	300:
		stAxis[GVL.cXP].mcMoveAbs(Axis:=stAxis[GVL.cXP].axisRef, Execute:=FALSE);
		stAxis[GVL.cXM].mcMoveAbs(Axis:=stAxis[GVL.cXM].axisRef, Execute:=FALSE);
		stAxis[GVL.cXP].mcMoveRel(Axis:=stAxis[GVL.cXP].axisRef, Execute:=FALSE);
		stAxis[GVL.cXM].mcMoveRel(Axis:=stAxis[GVL.cXM].axisRef, Execute:=FALSE);
		stAxis[GVL.cXP].mcJog(Axis:=stAxis[GVL.cXP].axisRef, JogForward:=FALSE, JogBackwards:=FALSE);
		stAxis[GVL.cXM].mcJog(Axis:=stAxis[GVL.cXM].axisRef, JogForward:=FALSE, JogBackwards:=FALSE);
		nNextState := 400;
		
	400:
		stAxis[GVL.cXP].mcReset(axis:=stAxis[GVL.cXP].axisRef, Execute:=TRUE);
		stAxis[GVL.cXM].mcReset(axis:=stAxis[GVL.cXM].axisRef, Execute:=TRUE);
		IF stAxis[GVL.cXP].mcReset.Done AND stAxis[GVL.cXM].mcReset.Done THEN
			stAxis[GVL.cXP].mcReset(axis:=stAxis[GVL.cXP].axisRef, Execute:=FALSE);
			stAxis[GVL.cXM].mcReset(axis:=stAxis[GVL.cXM].axisRef, Execute:=FALSE);
			bResetting := FALSE;
			nNextState := 100;
		END_IF
		//d := d+1;

END_CASE

END_FUNCTION_BLOCK

// ---- POUs/StateMachine/StateTop/FB_StateDisabled.TcPOU
FUNCTION_BLOCK FB_StateDisabled
VAR_IN_OUT
	stAxis  : ARRAY [GVL.cXP .. GVL.cXM] OF ST_AxisGroup;
	bTopentry : BOOL;
END_VAR
VAR_OUTPUT
	nSMState	: DINT;
END_VAR
VAR_INPUT

END_VAR

IF bTopEntry = TRUE THEN
	bTopEntry := FALSE;
END_IF	
	
stAxis[GVL.cXP].mcPower(Axis := stAxis[GVL.cXP].axisRef, Enable_Positive := FALSE, Enable_Negative := FALSE);
stAxis[GVL.cXM].mcPower(Axis := stAxis[GVL.cXM].axisRef, Enable_Positive := FALSE, Enable_Negative := FALSE);	
stAxis[GVL.cXP].mcHome(Axis := stAxis[GVL.cXP].axisRef, Execute := FALSE);
stAxis[GVL.cXM].mcHome(Axis := stAxis[GVL.cXP].axisRef, Execute := FALSE);
stAxis[GVL.cXP].mcReset(Axis := stAxis[GVL.cXP].axisRef, Execute := FALSE);
stAxis[GVL.cXM].mcReset(Axis := stAxis[GVL.cXM].axisRef, Execute := FALSE);
stAxis[GVL.cXP].bBrake 	:= GVL.cBrakeOn;
stAxis[GVL.cXM].bBrake 	:= GVL.cBrakeOn;
GVL.fbWaitTimer(IN:=FALSE);

nSMState := 10000;

END_FUNCTION_BLOCK

// ---- POUs/FB_Power.TcPOU
FUNCTION_BLOCK FB_Power

VAR_IN_OUT
	state : INT;
END_VAR

VAR
	//Power variable
	Vraw AT %I*	: ARRAY [0 .. E_Components.system] OF DINT;
	Vsense		: ARRAY [0 .. E_Components.system] OF REAL;
	Iin			: ARRAY [0 .. E_Components.system] OF REAL;
	Pin		 	: ARRAY [0 .. E_Components.system] OF REAL;
	Pin_max		: ARRAY [0 .. E_Components.system] OF REAL;
	Pin_avg		: ARRAY [0 .. E_Components.system] OF REAL;
	
	//counter
	i 				: INT;
	powerTotal		: ARRAY [0 .. E_Components.system] OF REAL;
	powerCounter 	: ARRAY [0 .. E_Components.system] OF DINT;
	
	//timer
	timer 			: TON;
	timeElapsed		: TIME;
	timer_rtrig		: R_TRIG;
	
	//testvar
	test : INT;
END_VAR

VAR CONSTANT
	Rsense			: REAL := 0.051;
	AdcResolution	: DINT := 8388607; //24bit adc (positive and minus)
	Vin				: ARRAY[0..1] OF REAL := [24.0, 48.0];
	Vref			: REAL := 1.25;
	CountTo			: TIME := T#1000H;
END_VAR

(*This function block is used to monitor shutter system power usage.
The module calculates instantanuous power, average power usage over a motion duration, and max power  *)

//reset power values
IF state=0 THEN
	FOR i := 0 TO E_Components.system BY 1 DO
		Pin_max[i] := 0;
	END_FOR
END_IF


FOR i:=0 TO (E_Components.system - 1) BY 1 DO 

//Calculate instantanuous power
	Vsense[i] := (DINT_TO_REAL(Vraw[i])*Vref)/DINT_TO_REAL(AdcResolution);
	Iin[i] := Vsense[i]/Rsense;
	
	IF i=E_Components.motorXM OR i=E_Components.motorXP THEN
		Pin[i] := Vin[1]*Iin[i];
	ELSE
		Pin[i] := Vin[0]*Iin[i];
	END_IF

	
//Calculate average power
	IF state <> 100 THEN
		powerTotal[i] := powerTotal[i]+Pin[i];
		powerCounter[i] := powerCounter[i]+1;
		Pin_avg[i] 		:= PowerTotal[i]/DINT_TO_REAL(powerCounter[i]);
	ELSE
			powertotal[i] 	:= 0;
			powerCounter[i]	:= 0;	
	END_IF

	
//Calculate max power
	IF Pin_max[i] < Pin[i] THEN
		Pin_max[i] := Pin[i];
	END_IF
	
END_FOR


//Calculate power of entire shutter
Pin[E_Components.system] := Pin[E_Components.motorXP]+Pin[E_Components.motorXM]+Pin[E_Components.brakes]
								+ Pin[E_Components.controller]+Pin[E_Components.terminals];
Pin_avg[E_Components.system] := Pin_avg[E_Components.motorXP]+Pin_avg[E_Components.motorXM]+Pin_avg[E_Components.brakes]
								+ Pin_avg[E_Components.controller]+Pin_avg[E_Components.terminals];
IF Pin_max[E_Components.system] < Pin[E_Components.system] THEN
	Pin_max[E_Components.system] := Pin[E_Components.system];
END_IF

END_FUNCTION_BLOCK

// ---- POUs/FB_Protection.TcPOU
FUNCTION_BLOCK FB_Protection
VAR_IN_OUT
	stAxis  			: ARRAY [GVL.cXP .. GVL.cXM] OF ST_AxisGroup;
	eCommand 			: E_Commands;
	//communication IN
	inCalibrate 		: ST_Calibrate;			// no protection needed
	inChangeAxisEnable	: ST_ChangeAxisEnable;	// no protection needed
	inChangeBrakeState	: ST_ChangeBrakeState;	// no protection needed
	inClearAllFaults	: ST_ClearAllFaults;	// no protection needed
	inClearAxisFaults	: ST_ClearAxisFaults;	// no protection needed
	inCloseShutter		: ST_CloseShutter;		
	inDisableAllAxes	: ST_DisableAllAxes;
	inEnableAllAxes		: ST_EnableAllAxes;
	inGoToProd			: ST_GoToProd;
	inHomeAxis			: ST_HomeAxis;
	inMoveAxisAbsolute	: ST_MoveAxisAbsolute;
	inMoveAxisRelative	: ST_MoveAxisRelative;
	inOpenShutter		: ST_OpenShutter;
	inReset				: ST_Reset;
	inTakeExposure		: ST_TakeExposure;
	inToggleSafetyCheck	: ST_ToggleSafetyCheck;
END_VAR
VAR_INPUT
	nState 			: DINT;
END_VAR
VAR_OUTPUT
	nShutterError	: UINT;
END_VAR
VAR
	checkHomed_TON 	: TON;
	
	//for use end of travel protection
	fEotDistTravel	: ARRAY [GVL.cXP .. GVL.cXM, cLmHome .. cLmDeploy] OF LREAL;
	fEotDistStart	: ARRAY [GVL.cXP .. GVL.cXM, cLmHome .. cLmDeploy] OF LREAL;
	fbEotRtrig		: ARRAY [GVL.cXP .. GVL.cXM, cLmHome .. cLmDeploy] OF R_Trig;
	
	//other Var
	i	: INT;
	bBadHall : BOOL;
END_VAR

VAR CONSTANT
	cLmHome 		: INT 	:= 0;
	cLmDeploy		: INT 	:= 1;
	cEotTravelLm	: LREAL := 1.5;
	cDiffLimit 		: LREAL	:= 5;
	cPosError		: LREAL	:= 0.3;
	cExpoTimer		: TIME	:= T#100MS;
	cMaxVelocity	: LREAL	:= 1668.355556;
	cMinVelocity	: LREAL	:= 0;
END_VAR

(*
This function block contains the logic for the shutter system protection. 
*)
/////////////////////////////////////////////////////////////////////////////////////////////////////////////////////
(*Reset Errors*)
/////////////////////////////////////////////////////////////////////////////////////////////////////////////////////
IF (eCommand=E_Commands.reset) THEN
	stAxis[GVL.cXP].fPosDiffAtTrip 		:= 0;
	stAxis[GVL.cXM].fPosDiffAtTrip 		:= 0;
	fEotDistStart[GVL.cXP,cLmHome] 		:= stAxis[GVL.cXP].axisRef.NcToPlc.ActPos;
	fEotDistStart[GVL.cXP,cLmDeploy] 	:= stAxis[GVL.cXP].axisRef.NcToPlc.ActPos;
	fEotDistStart[GVL.cXM,cLmHome] 		:= stAxis[GVL.cXM].axisRef.NcToPlc.ActPos;
	fEotDistStart[GVL.cXM,cLmDeploy] 	:= stAxis[GVL.cXM].axisRef.NcToPlc.ActPos;
	nShutterError 						:= 0;
END_IF
IF (eCommand=E_Commands.calibrate) THEN
	bBadHall := FALSE;
END_IF

nShutterError.0 := 0;

/////////////////////////////////////////////////////////////////////////////////////////////////////////////////////
(*Check brake status - prevents motion if motion is commanded while brake is engaged*)
/////////////////////////////////////////////////////////////////////////////////////////////////////////////////////
IF stAxis[GVL.cXP].bBrake = GVL.cBrakeOn OR stAxis[GVL.cXM].bBrake = GVL.cBrakeOn THEN
	IF stAxis[GVL.cXP].axisRef.Status.Moving OR stAxis[GVL.cXM].axisRef.Status.Moving THEN
		//////// --set error here-- //////////////////////////////////////////////////////////////////////////////////////////
		nShutterError.1 := 1;
	ELSE
		nShutterError.1 := 0;
	END_IF
END_IF

/////////////////////////////////////////////////////////////////////////////////////////////////////////////////////
(*Check position differences - Compare hall switch and motor encoder position. Stop motion if greater than diffLimit.*)
/////////////////////////////////////////////////////////////////////////////////////////////////////////////////////
IF stAxis[GVL.cXP].bIsCalibrated AND stAxis[GVL.cXM].bIsCalibrated THEN
	IF ABS(stAxis[GVL.cXP].fPosDiffAtTrip)>cDiffLimit OR ABS(stAxis[GVL.cXM].fPosDiffAtTrip)>cDiffLimit THEN
		//////// --set error here-- /////////////////////////////////////////////////////////////////////////////////
		nShutterError.2 := 1;
	ELSE
		nShutterError.2 := 0;
	END_IF
END_IF

/////////////////////////////////////////////////////////////////////////////////////////////////////////////////////
(*Check exposure time - If less than 100 ms, prevent exposure command from running*)
/////////////////////////////////////////////////////////////////////////////////////////////////////////////////////
IF (inTakeExposure.exposureTime<cExpoTimer AND eCommand=E_Commands.takeExposure) THEN
	eCommand := E_Commands.noCommand;
	//////// --set error here-- /////////////////////////////////////////////////////////////////////////////////
	nShutterError.3 := 1;
ELSE
	nShutterError.3 := 0;
END_IF

/////////////////////////////////////////////////////////////////////////////////////////////////////////////////////
(*Check home status - Prevents all other motion if not homed*)
/////////////////////////////////////////////////////////////////////////////////////////////////////////////////////
IF NOT stAxis[GVL.cXP].axisRef.Status.Homed OR NOT stAxis[GVL.cXM].axisRef.Status.Homed THEN
	IF eCommand=E_Commands.closeShutter OR eCommand=E_Commands.goToProd 
		OR eCommand=E_Commands.moveAxisAbsolute OR eCommand=E_Commands.moveAxisRelative 
		OR eCommand=E_Commands.openShutter OR eCommand=E_Commands.takeExposure THEN
			//////// --set error here-- /////////////////////////////////////////////////////////////////////////////////
			nShutterError.4 := 1;
	END_IF
ELSE
	nShutterError.4 := 0;
END_IF
/////////////////////////////////////////////////////////////////////////////////////////////////////////////////////
(*Check for NC errors. If any, disable movement for both motors*)
/////////////////////////////////////////////////////////////////////////////////////////////////////////////////////
IF stAxis[GVL.cXP].axisRef.Status.Error OR stAxis[GVL.cXM].axisRef.Status.Error THEN
	stAxis[GVL.cXP].mcPower(Axis := stAxis[GVL.cXP].axisRef, Enable_Positive := FALSE, Enable_Negative := FALSE);
	stAxis[GVL.cXM].mcPower(Axis := stAxis[GVL.cXM].axisRef, Enable_Positive := FALSE, Enable_Negative := FALSE); 
	stAxis[GVL.cXP].bBrake := GVL.cBrakeOn;
	stAxis[GVL.cXM].bBrake := GVL.cBrakeOn;
	//////// --set error here-- /////////////////////////////////////////////////////////////////////////////////
	nShutterError.5 := 1;
ELSE
	nShutterError.5 := 0;
END_IF

/////////////////////////////////////////////////////////////////////////////////////////////////////////////////////
(*Check calibration status - If one blade set is not calibrated, speed cannot be higher than 200 mms.*)
/////////////////////////////////////////////////////////////////////////////////////////////////////////////////////
IF NOT stAxis[GVL.cXP].bIsCalibrated OR NOT stAxis[GVL.cXM].bIsCalibrated THEN
	IF (inMoveAxisAbsolute.speed>200) THEN
		inMoveAxisAbsolute.speed := 0;
		//////// --set error here-- /////////////////////////////////////////////////////////////////////////////////
		nShutterError.6 := 1;
	END_IF
ELSE
	nShutterError.6:= 0;
END_IF

/////////////////////////////////////////////////////////////////////////////////////////////////////////////////////
(*Check that one blade set cannot be commanded to pass limit*)
/////////////////////////////////////////////////////////////////////////////////////////////////////////////////////
IF (eCommand=E_Commands.moveAxisAbsolute AND (stAxis[GVL.cXP].axisRef.Status.Homed AND stAxis[GVL.cXM].axisRef.Status.Homed)) THEN
	IF (inMoveAxisAbsolute.position<(GVL.cPosStart-cPosError) OR inMoveAxisAbsolute.position>(GVL.cPosEnd+cPosError)) THEN
		eCommand := E_Commands.noCommand;
		//////// --set error here-- /////////////////////////////////////////////////////////////////////////////////
		nShutterError.7 := 1;
	END_IF
END_IF
IF (eCommand=E_Commands.moveAxisRelative AND (stAxis[GVL.cXP].axisRef.Status.Homed AND stAxis[GVL.cXM].axisRef.Status.Homed)) THEN
	IF ((inMoveAxisRelative.distance+stAxis[inMoveAxisRelative.axisIndex].axisRef.NcToPlc.ActPos)<(GVL.cPosStart-cPosError) 
		OR (inMoveAxisRelative.distance+stAxis[inMoveAxisRelative.axisIndex].axisRef.NcToPlc.ActPos)>(GVL.cPosEnd+cPosError)) THEN
		eCommand := E_Commands.noCommand;
		//////// --set error here-- /////////////////////////////////////////////////////////////////////////////////
		nShutterError.7 := 1;
	END_IF
END_IF

/////////////////////////////////////////////////////////////////////////////////////////////////////////////////////
(*Check that one blade set cannot be commanded to pass the other blade set's position*)
/////////////////////////////////////////////////////////////////////////////////////////////////////////////////////
IF (eCommand=E_Commands.moveAxisAbsolute) THEN
	IF (inMoveAxisAbsolute.axisIndex=GVL.cXP AND inMoveAxisAbsolute.position>(stAxis[GVL.cXM].axisRef.NcToPlc.ActPos+cPosError)) THEN
		eCommand := E_Commands.noCommand;
		//////// --set error here-- /////////////////////////////////////////////////////////////////////////////////
		nShutterError.8 := 1;
	END_IF
	IF (inMoveAxisAbsolute.axisIndex=GVL.cXM AND inMoveAxisAbsolute.position<(stAxis[GVL.cXP].axisRef.NcToPlc.ActPos-cPosError)) THEN
		eCommand := E_Commands.noCommand;
		//////// --set error here-- /////////////////////////////////////////////////////////////////////////////////
		nShutterError.8 := 1;
	END_IF
END_IF

IF (eCommand=E_Commands.moveAxisRelative) THEN
	IF (inMoveAxisRelative.axisIndex=GVL.cXP AND (inMoveAxisRelative.distance+stAxis[GVL.cXP].axisRef.NcToPlc.ActPos)>(stAxis[GVL.cXM].axisRef.NcToPlc.ActPos+cPosError)) THEN
		eCommand := E_Commands.noCommand;
		//////// --set error here-- /////////////////////////////////////////////////////////////////////////////////
		nShutterError.8 := 1;
	END_IF
	IF (inMoveAxisRelative.axisIndex=GVL.cXM AND (inMoveAxisRelative.distance+stAxis[GVL.cXM].axisRef.NcToPlc.ActPos)<(stAxis[GVL.cXP].axisRef.NcToPlc.ActPos-cPosError)) THEN
		eCommand := E_Commands.noCommand;
		//////// --set error here-- /////////////////////////////////////////////////////////////////////////////////
		nShutterError.8 := 1;
	END_IF
END_IF

/////////////////////////////////////////////////////////////////////////////////////////////////////////////////////
(* Checks to see if blades have reach end of travel. If it has, stop further motion in that direction	*)
/////////////////////////////////////////////////////////////////////////////////////////////////////////////////////
//End of travel stop
IF(stAxis[GVL.cXP].axisRef.Status.Homed AND stAxis[GVL.cXM].axisRef.Status.Homed) THEN
	fbEotRtrig[GVL.cXP,cLmHome](CLK := stAxis[GVL.cXP].bLimitHome);
	fbEotRtrig[GVL.cXP,cLmDeploy](CLK := stAxis[GVL.cXP].bLimitDeployed);
	fbEotRtrig[GVL.cXM,cLmHome](CLK := stAxis[GVL.cXM].bLimitHome);
	fbEotRtrig[GVL.cXM,cLmDeploy](CLK := stAxis[GVL.cXM].bLimitDeployed);
	IF fbEotRtrig[GVL.cXP,cLmHome].Q THEN
		fEotDistStart[GVL.cXP,cLmHome] := stAxis[GVL.cXP].axisRef.NcToPlc.ActPos;
	END_IF
	IF fbEotRtrig[GVL.cXP,cLmDeploy].Q THEN
		fEotDistStart[GVL.cXP,cLmDeploy] := stAxis[GVL.cXP].axisRef.NcToPlc.ActPos;
	END_IF
	IF fbEotRtrig[GVL.cXM,cLmHome].Q THEN
		fEotDistStart[GVL.cXM,cLmHome] := stAxis[GVL.cXM].axisRef.NcToPlc.ActPos;
	END_IF
	IF fbEotRtrig[GVL.cXM,cLmDeploy].Q THEN
		fEotDistStart[GVL.cXM,cLmDeploy] := stAxis[GVL.cXM].axisRef.NcToPlc.ActPos;
	END_IF									
	
	IF stAxis[GVL.cXP].bLimitHome THEN
		fEotDistTravel[GVL.cXP,cLmHome] := fEotDistStart[GVL.cXP,cLmHome] - stAxis[GVL.cXP].axisRef.NcToPlc.ActPos;
		IF fEotDistTravel[GVL.cXP,cLmHome] > cEotTravelLm THEN
			stAxis[GVL.cXP].mcPower(Axis := stAxis[GVL.cXP].axisRef, Enable_Negative := FALSE);
		END_IF
	END_IF
	
	IF stAxis[GVL.cXP].bLimitDeployed THEN
		fEotDistTravel[GVL.cXP,cLmDeploy] := stAxis[GVL.cXP].axisRef.NcToPlc.ActPos - fEotDistStart[GVL.cXP,cLmDeploy];
		IF fEotDistTravel[GVL.cXP,cLmHome] > cEotTravelLm THEN
			stAxis[GVL.cXP].mcPower(Axis := stAxis[GVL.cXP].axisRef, Enable_Positive := FALSE);
		END_IF
	END_IF
	
	IF stAxis[GVL.cXM].bLimitHome THEN
		fEotDistTravel[GVL.cXM,clmHome] := stAxis[GVL.cXM].axisRef.NcToPlc.ActPos - fEotDistStart[GVL.cXM,cLmHome];
		IF fEotDistTravel[GVL.cXM,cLmHome] > cEotTravelLm THEN
			stAxis[GVL.cXM].mcPower(Axis := stAxis[GVL.cXM].axisRef, Enable_Positive := FALSE);
		END_IF
	END_IF
	
	IF stAxis[GVL.cXM].bLimitDeployed THEN
		fEotDistTravel[GVL.cXM,cLmDeploy] := fEotDistStart[GVL.cXM,cLmDeploy] - stAxis[GVL.cXM].axisRef.NcToPlc.ActPos;
		IF fEotDistTravel[GVL.cXM,cLmHome] > cEotTravelLm THEN
			stAxis[GVL.cXM].mcPower(Axis := stAxis[GVL.cXM].axisRef, Enable_Negative := FALSE);
		END_IF
	END_IF
END_IF

/////////////////////////////////////////////////////////////////////////////////////////////////////////////////////
(* if hall signal changes during no motion, system needs to recalibrate	*)
/////////////////////////////////////////////////////////////////////////////////////////////////////////////////////
FOR i:=GVL.cHallLower TO GVL.cHallUpper BY 1 DO
	IF GVL.nNumOfInputs[i].0 AND ((NOT stAxis[GVL.cXP].axisRef.Status.Moving) AND (NOT stAxis[GVL.cXM].axisRef.Status.Moving)) THEN
		bBadHall := TRUE;
	END_IF
END_FOR
IF bBadHall THEN
	IF eCommand=E_Commands.closeShutter OR eCommand=E_Commands.goToProd 
		OR eCommand=E_Commands.moveAxisAbsolute OR eCommand=E_Commands.moveAxisRelative 
		OR eCommand=E_Commands.openShutter OR eCommand=E_Commands.takeExposure THEN
			nShutterError.13 := 1;
	END_IF
END_IF

/////////////////////////////////////////////////////////////////////////////////////////////////////////////////////
(* shutter system error handle	*)
/////////////////////////////////////////////////////////////////////////////////////////////////////////////////////

IF (nShutterError.0 OR_ELSE nShutterError.1 OR_ELSE nShutterError.2 OR_ELSE nShutterError.3 OR_ELSE nShutterError.4 OR_ELSE nShutterError.5) THEN
	stAxis[GVL.cXP].mcStop(Axis := stAxis[GVL.cXP].axisRef, Deceleration := 29630, Jerk := 263374.5, Execute := TRUE);
	stAxis[GVL.cXM].mcStop(Axis := stAxis[GVL.cXM].axisRef, Deceleration := 29630, Jerk := 263374.5, Execute := TRUE);
	//stAxis[GVL.cXP].mcPower(Axis := stAxis[GVL.cXP].axisRef, Enable_Positive := FALSE, Enable_Negative := FALSE);
	//stAxis[GVL.cXM].mcPower(Axis := stAxis[GVL.cXM].axisRef, Enable_Positive := FALSE, Enable_Negative := FALSE); 
	IF (nShutterError.0 OR_ELSE nShutterError.2 OR_ELSE nShutterError.3 OR_ELSE nShutterError.4 OR_ELSE nShutterError.5 OR_ELSE nShutterError.13) THEN
		stAxis[GVL.cXP].bBrake := GVL.cBrakeOn;
		stAxis[GVL.cXM].bBrake := GVL.cBrakeOn;
	END_IF
ELSE
	stAxis[GVL.cXP].mcStop(Axis := stAxis[GVL.cXP].axisRef, Execute := FALSE);
	stAxis[GVL.cXM].mcStop(Axis := stAxis[GVL.cXM].axisRef, Execute := FALSE);
END_IF

/////////////////////////////////////////////////////////////////////////////////////////////////////////////////////
(* Other shutter protection	*)
/////////////////////////////////////////////////////////////////////////////////////////////////////////////////////

//Min and Max speed for PROD
IF (inReset.speed>cMaxVelocity) THEN
	inReset.speed:=cMaxVelocity;
ELSIF (inReset.speed<cMinVelocity) THEN
	inReset.speed:=cMinVelocity;
END_IF
//Min and Max speed for move absolute
IF (inMoveAxisAbsolute.speed>cMaxVelocity) THEN
	inReset.speed:=cMaxVelocity;
ELSIF (inMoveAxisAbsolute.speed<cMinVelocity) THEN
	inReset.speed:=cMinVelocity;
END_IF

END_FUNCTION_BLOCK

// ---- POUs/StateMachine/FB_Tracking.TcPOU
FUNCTION_BLOCK FB_Tracking
VAR_IN_OUT
	stAxis  : ARRAY [GVL.cXP .. GVL.cXM] OF ST_AxisGroup;	
END_VAR
VAR_INPUT
	eCommand 			: E_Commands;
	bMotionDone			: BOOL;
	inReset				: ST_Reset;
	inMoveAxisAbsolute	: ST_MoveAxisAbsolute;
	inMoveAxisRelative	: ST_MoveAxisRelative;
END_VAR
VAR_OUTPUT
	stOutMotionDone : ST_MotionDone;
END_VAR
VAR
	//used in tracking Action
	stTrack			: ARRAY [0 .. 4] OF ST_TRACK;
	stTrackTemp		: ST_TRACK;  // Used for the sorting of stTrack.
	keepSorting		: BOOL;      // Used for the sorting.
	bGoNextSeq		: BOOL;
	nAxisID			: INT;
	nMask			: ULINT := 16#FFFF_FFFF_0000_0000;
	
	//used in determining target duration
	fSpeed			: LREAL;
	tTargetDur		: LTIME;
	fDistance		: LREAL;
	
	fbMoving_Rtrig : ARRAY[0 .. 1] OF R_TRIG;
	fbRtrig		: ARRAY[GVL.cHallLower..GVL.cHallUpper] OF R_Trig;
	bInMotion	: BOOL;
	stMotionDone : ARRAY [0..1] OF ST_MotionDone;	
	nSequence	: DINT;
	nLastMoved	: INT;
	
	//counter
	i, j, k, m		: INT := 0;
	nTPC	: INT; //Trip Per Cycle

	// Save task-start and MIO SysTime values in a ring buffer x of depth N. The newest
	// entry is x[i], the oldest is x[(i + 1) mod N], assuming that the buffer is full.
	iTimeBuffer: INT := GVL.cTimeBufferDepth - 1;
	taskStartExtTime: T_TaskStartTimes;
	mioSysTime: T_MioSysTimes;

END_VAR

//////////////////////////////////////////////////////////////
// Call this function block once per cycle to process any updated information about blade set motion and send updates to CCS if required.
//////////////////////////////////////////////////////////////

// Update some times for the previous and current cycles.
iTimeBuffer := (iTimeBuffer + 1) MOD GVL.cTimeBufferDepth;
taskStartExtTime[iTimeBuffer] := F_GetCurExtTime64(GVL.DcToExtTimeOffset, GVL.DcToTcTimeOffset);
mioSysTime[iTimeBuffer] := GVL.mioSysTime;

stAxis[GVL.cXP].bTrackedFlag:=FALSE;
stAxis[GVL.cXM].bTrackedFlag:=FALSE;
nTPC:=0;

// Detect start of motion for the +X blade set, rising edge of its Moving flag from the motor controller.
// Reset motion profile parameters in a local motion-done message not monitored by CCS.
fbMoving_Rtrig[GVL.cXP](CLK:=stAxis[GVL.cXP].axisRef.Status.Moving);
IF fbMoving_Rtrig[GVL.cXP].Q THEN
	// Prepare to record motion profile information.
	bInMotion:=TRUE;  // We're moving!
	stMotionDone[GVL.cXP].axisNum := GVL.cXP; // Axis is +X.
	stMotionDone[GVL.cXP].nsamples := 0;      // No encoder samples yet.
	stMotionDone[GVL.cXP].ntrans := 0;        // No Hall transitions yet.
	stMotionDone[gvl.cXP].startPos := stAxis[GVL.cXP].axisRef.NcToPlc.ActPos;   // Where are we now?
	stMotionDone[GVL.cXP].startTime := taskStartExtTime[iTimeBuffer];
	stMotionDone[GVL.cXP].targetDur := LTIME#0D0H0M0S0MS0US0NS;  // Don't know yet how long this motion will take.
END_IF

// The same, but for the -X blade set.
fbMoving_Rtrig[GVL.cXM](CLK:=stAxis[GVL.cXM].axisRef.Status.Moving);
IF fbMoving_Rtrig[GVL.cXM].Q THEN
	// Prepare to record motion profile information.
	bInMotion:=TRUE;
	stMotionDone[gvl.cXM].axisNum := GVL.cXM;
	stMotionDone[gvl.cXM].nsamples := 0;
	stMotionDone[gvl.cXM].ntrans := 0;
	stMotionDone[gvl.cXM].startPos := stAxis[GVL.cXM].axisRef.NcToPlc.ActPos;
	stMotionDone[gvl.cXM].startTime := taskStartExtTime[iTimeBuffer];
	stMotionDone[gvl.cXM].targetDur := LTIME#0D0H0M0S0MS0US0NS;
END_IF

// Assuming that a motion command was issued by CCS, calculate how long the motion is supposed to last.
// Output is tTargetDur.
IF eCommand = E_Commands.takeExposure THEN
	fSpeed	:= inReset.speed;   // Speed from reset command (actually now set elsewhere in this PLC code).
	IF (fSpeed>0) THEN
		IF (fSpeed>1668.355556) THEN
			fSpeed:=1668.355556;
		END_IF
		tTargetDur 	:= LREAL_TO_LTIME((2*GVL.cPosEnd)/(fSpeed)*EXPT(10,9));
	END_IF
ELSIF eCommand = E_Commands.moveAxisAbsolute THEN
	// MoveAxisAbsolute message contains target position and speed of motion.
	fDistance := ABS(stAxis[inMoveAxisAbsolute.axisIndex].axisRef.NcToPlc.ActPos - inMoveAxisAbsolute.position);
	fSpeed	:= inMoveAxisAbsolute.speed;
	IF (fSpeed>0) THEN
		IF (fSpeed>1668.355556) THEN
			fSpeed:=1668.355556;
		END_IF
		tTargetDur 	:= LREAL_TO_LTIME(((2*fDistance)/(fSpeed))*EXPT(10,9));
	END_IF
ELSIF eCommand = E_Commands.moveAxisRelative THEN
	// MoveAxisRelative message contains position change and how long to take to do it.
	tTargetDur	:= TIME_TO_LTIME(inMoveAxisRelative.moveTime);
END_IF

//Checks to see which blade set last started moving.
IF (stAxis[GVL.cXM].axisRef.Status.Moving AND stAxis[GVL.cXP].axisRef.Status.InTargetPosition) THEN
	nLastMoved:=GVL.cXM;
ELSIF (stAxis[GVL.cXP].axisRef.Status.Moving AND stAxis[GVL.cXM].axisRef.Status.InTargetPosition) THEN
	nLastMoved:=GVL.cXP;
END_IF

////////// Handle the completion of a blade set motion. //////////
IF bMotionDone THEN
	//use for determining which blade set has finished during a travelling slit motion
	IF (stAxis[GVL.cXM].axisRef.Status.Moving AND stAxis[GVL.cXP].axisRef.Status.InTargetPosition) THEN
		nAxisID:=GVL.cXP;
	ELSIF (stAxis[GVL.cXP].axisRef.Status.Moving AND stAxis[GVL.cXM].axisRef.Status.InTargetPosition) THEN
		nAxisID:=GVL.cXM;
	ELSE 
		nAxisID:=nLastMoved;
	END_IF
	//bInMotion flag remains true if either of the blade sets is still in motion
	IF ((NOT stAxis[GVL.cXP].axisRef.Status.Moving) AND (NOT stAxis[GVL.cXM].axisRef.Status.Moving)) THEN
		bInMotion := FALSE;
	END_IF
	// Complete our local motion-done message.
	nSequence := nSequence+1;
	// The motor controller doesn't report exactly when motion was completed, so we assume that it was when the process data
	// from the controller reached us, i.e., at the start of the current cycle.
	stMotionDone[nAxisID].actualDur := ULINT_TO_LTIME(taskStartExtTime[iTimeBuffer] - stMotionDone[nAxisID].startTime);
	stMotionDone[nAxisID].targetDur := tTargetDur;
	stMotionDone[nAxisID].targetPos := stAxis[nAxisID].axisRef.NcToPlc.TargetPos;
	stMotionDone[nAxisID].endPos := stAxis[nAxisID].axisRef.NcToPlc.ActPos;
	stMotionDone[nAxisId].ptpState := MAIN.ptpDiagInfo.PTPState;
	stMotionDone[nAxisId].leapSeconds := MAIN.ptpDiagInfo.CurrentUtcOffset;
	stMotionDone[nAxisId].leapIsValid := TO_BOOL(MAIN.ptpDiagInfo.CurrentUtcOffsetIsValid);
	// Copy our local motion-done message to the location that's monitored by CCS.
	stOutMotionDone:=stMotionDone[nAxisID];
	stOutMotionDone.sequence:=nSequence;  // Ensure message gets sent to CCS by making sure that at least one field has a changed value.
END_IF


////////// Collect information on any Hall switch transitions from the MIOs. //////////
// nNumOfINputs[i] is linked to the event count for the MIO channel assigned to Hall sensor i.
// bInputEventState[i] is linked to the current MIO channel state for Hall sensor i.
// nInputEventTime[i] is linked to the first transition timestamp for Hall sensor i. We assume there is at most one per cycle per channel, though
// more than one channel may have a timestamp available in the same cycle.
// New timestamps are added to the end of the stTrack array.

FOR i:=GVL.cHallLower TO GVL.cHallUpper BY 1 DO
	fbRtrig[i](CLK:=GVL.nNumOfInputs[i].0);  // Look for a rising edge in channel status, which means we have a transition timestamp.
	IF fbRtrig[i].Q THEN
		stTrack[nTPC].nSeqToCompare := INT_TO_WORD((i*10)+5);
		stTrack[nTPC].bEdgeToCompare := GVL.bInputEventState[i];
		stTrack[nTPC].nHallID := i;
		stTrack[nTPC].tScanTime := 
			F_MioExtTime(i, GVL.nInputEventTime[i], iTimeBuffer, taskStartExtTime, mioSysTime);  // ADC timestamp -> ext time.
 		// Count the number of entries stored in stTrack.
		nTPC:=nTPC+1;
	END_IF
END_FOR
	
// Calibration stores events in time order, and later code that assigns locations to Hall events requires
// exactly the same ordering for a given blade set and direction of motion. If during this cycle we picked up
// events from more than one channel we'll have to sort them by time. At most a handful of events
// may occur in a cycle so an exchange sort will do.
IF nTPC > 1 THEN
	keepSorting := TRUE;  // Do we need to keep sorting?
	WHILE keepSorting DO
		keepSorting := FALSE;
		FOR j:= nTPC - 1 TO 1 BY -1 DO
			IF (stTrack[j].tScanTime < stTrack[j-1].tScanTime) THEN  // Use <, not <=, to make it a stable sort.
				stTrackTemp := stTrack[j];
				stTrack[j] := stTrack[j-1];
				stTrack[j-1] := stTrackTemp;
				keepSorting := TRUE;  // Need to keep sorting if an exchange was made.
			END_IF
		END_FOR
	END_WHILE
END_IF


// If we picked up some Hall transitions this cycle, then we need to take position samples (encoder readout).
// We want to check if the position of a blade set at the time of a Hall transition agrees with the
// Hall switch position taken from the last calibration.
IF nTPC>0 THEN
	FOR k:=0 TO nTPC-1 BY 1 DO
		IF (stAxis[GVL.cXP].axisRef.Status.Moving AND stAxis[GVL.cXM].axisRef.Status.Moving) AND
			(stAxis[GVL.cXP].axisRef.Status.PositiveDirection AND stAxis[GVL.cXM].axisRef.Status.PositiveDirection) THEN
			ACT_TrackingDoublePositive();
		ELSIF (stAxis[GVL.cXP].axisRef.Status.Moving AND stAxis[GVL.cXM].axisRef.Status.Moving) AND
			(stAxis[GVL.cXP].axisRef.Status.NegativeDirection AND stAxis[GVL.cXM].axisRef.Status.NegativeDirection) THEN
			ACT_TrackingDoubleNegative();
		ELSE
			ACT_TrackingSingle();
		END_IF
		bGoNextSeq:=FALSE;
	END_FOR
END_IF

ACTION ACT_TrackingDoubleNegative:
// Take encoder samples and compare against Hall transitions when both blade sets are moving toward decreasing camera X coordinate.
// Remember, this code is being called from inside a loop over the contents of stTrack[] with k being the loop variable.
// We have to first assign a Hall event to a blade set before we can find out the motion start times and
// calculate elapsed times from that. 

// +X blade set
IF stAxis[GVL.cXP].axisRef.Status.Moving THEN
	//Compare current sequence with recorded sequence. Update position if match. Negative direction.
	IF stAxis[GVL.cXP].axisRef.status.NegativeDirection AND stAxis[GVL.cXP].stHall[GVL.cDirNeg, stAxis[GVL.cXP].nTripCount].nSeq = stTrack[k].nSeqToCompare AND
			stAxis[GVL.cXP].stHall[GVL.cDirNeg, stAxis[GVL.cXP].nTripCount].bEdge = stTrack[k].bEdgeToCompare AND (NOT bGoNextSeq) THEN
		stAxis[GVL.cXP].fHallPosAct := stAxis[GVL.cXP].fHallPosCal[GVL.cDirNeg, stAxis[GVL.cXP].nTripCount];
		stAxis[GVL.cXP].nTripCount := stAxis[GVL.cXP].nTripCount - 1;		
		//track difference between hall sensor and encoder data at trip point
		stAxis[GVL.cXP].fPosDiffAtTrip := stAxis[GVL.cXP].axisRef.NcToPlc.ActPos - stAxis[GVL.cXP].fHallPosAct;
		stAxis[GVL.cXP].bTrackedFlag:=TRUE;
		bGoNextSeq:=TRUE;
		
		IF bInMotion AND MAIN.outShutterStatus.smState<>E_StatesMaint.Calibrating THEN
			nAxisID := GVL.cXP;
			// The Hall event belongs to the +X blade set.
			stMotionDone[GVL.cXP].trans[stMotionDone[GVL.cXP].ntrans].extTime := stTrack[k].tScanTime;
			stMotionDone[GVL.cXP].trans[stMotionDone[GVL.cXP].ntrans].id := stTrack[k].nHallID;
			stMotionDone[GVL.cXP].trans[stMotionDone[GVL.cXP].ntrans].on := stTrack[k].bEdgeToCompare;
			stMotionDone[GVL.cXP].trans[stMotionDone[GVL.cXP].ntrans].pos := stAxis[GVL.cXP].fHallPosAct;
			stMotionDone[GVL.cXP].ntrans := stMotionDone[GVL.cXP].ntrans +1;
			// We're taking the encoder value from process data for this cycle, so the closest
			// approximation we have to the actual sample time is the time at the start of the cycle.
			stMotionDone[GVL.cXP].samples[stMotionDone[GVL.cXP].nsamples].extTime := taskStartExtTime[iTimeBuffer];
			stMotionDone[GVL.cXP].samples[stMotionDone[GVL.cXP].nsamples].pos := stAxis[GVL.cXP].axisRef.NcToPlc.ActPos;
			stMotionDone[GVL.cXP].nsamples := stMotionDone[GVL.cXP].nsamples + 1;
		END_IF
		
	END_IF
END_IF

// -X blade set
IF stAxis[GVL.cXM].axisRef.Status.Moving THEN
	//Compare current sequence with recorded sequence. Update position if match. Negative direction.
	IF stAxis[GVL.cXM].axisRef.status.NegativeDirection AND stAxis[GVL.cXM].stHall[GVL.cDirNeg, stAxis[GVL.cXM].nTripCount].nSeq = stTrack[k].nSeqToCompare AND
			stAxis[GVL.cXM].stHall[GVL.cDirNeg, stAxis[GVL.cXM].nTripCount].bEdge = stTrack[k].bEdgeToCompare AND (NOT bGoNextSeq) THEN
		stAxis[GVL.cXM].fHallPosAct := stAxis[GVL.cXM].fHallPosCal[GVL.cDirNeg, stAxis[GVL.cXM].nTripCount];
		stAxis[GVL.cXM].nTripCount := stAxis[GVL.cXM].nTripCount + 1;	
		//track difference between hall sensor and encoder data at trip point
		stAxis[GVL.cXM].fPosDiffAtTrip := stAxis[GVL.cXM].axisRef.NcToPlc.ActPos - stAxis[GVL.cXM].fHallPosAct;
		stAxis[GVL.cXM].bTrackedFlag:=TRUE;
		bGoNextSeq:=TRUE;
		
		IF bInMotion AND MAIN.outShutterStatus.smState<>E_StatesMaint.Calibrating THEN
			nAxisID:= GVL.cXM;
			// The Hall event belongs to the -X blade set.
			stMotionDone[GVL.cXM].trans[stMotionDone[GVL.cXM].ntrans].extTime := stTrack[k].tScanTime;
			stMotionDone[GVL.cXM].trans[stMotionDone[GVL.cXM].ntrans].id := stTrack[k].nHallID;
			stMotionDone[GVL.cXM].trans[stMotionDone[GVL.cXM].ntrans].on := stTrack[k].bEdgeToCompare;
			stMotionDone[GVL.cXM].trans[stMotionDone[GVL.cXM].ntrans].pos := stAxis[GVL.cXM].fHallPosAct;
			stMotionDone[GVL.cXM].ntrans := stMotionDone[GVL.cXM].ntrans +1;

			stMotionDone[GVL.cXM].samples[stMotionDone[GVL.cXM].nsamples].extTime := taskStartExtTime[iTimeBuffer];
			stMotionDone[GVL.cXM].samples[stMotionDone[GVL.cXM].nsamples].pos := stAxis[GVL.cXM].axisRef.NcToPlc.ActPos;
			stMotionDone[GVL.cXM].nsamples := stMotionDone[GVL.cXM].nsamples + 1;
		END_IF
		
	END_IF
END_IF
END_ACTION

ACTION ACT_TrackingDoublePositive:
// Take encoder samples and compare against Hall transitions when both blade sets are moving toward increasing camera X coordinate.

// -X blade set
IF stAxis[GVL.cXM].axisRef.Status.Moving THEN
	//Compare current sequence with recorded sequence. Update position if match. Positive direction.
	IF stAxis[GVL.cXM].axisRef.status.PositiveDirection AND stAxis[GVL.cXM].stHall[GVL.cDirPos, stAxis[GVL.cXM].nTripCount].nSeq = stTrack[k].nSeqToCompare AND
			stAxis[GVL.cXM].stHall[GVL.cDirPos, stAxis[GVL.cXM].nTripCount].bEdge = stTrack[k].bEdgeToCompare AND (NOT bGoNextSeq) THEN
		stAxis[GVL.cXM].fHallPosAct := stAxis[GVL.cXM].fHallPosCal[GVL.cDirPos, stAxis[GVL.cXM].nTripCount];
		stAxis[GVL.cXM].nTripCount := stAxis[GVL.cXM].nTripCount - 1;	
		//track difference between hall sensor and encoder data at trip point
		stAxis[GVL.cXM].fPosDiffAtTrip := stAxis[GVL.cXM].axisRef.NcToPlc.ActPos - stAxis[GVL.cXM].fHallPosAct;
		stAxis[GVL.cXM].bTrackedFlag:=TRUE;
		bGoNextSeq:=TRUE;
		
		IF bInMotion AND MAIN.outShutterStatus.smState<>E_StatesMaint.Calibrating THEN
			nAxisID:= GVL.cXM;
			// The Hall event belongs to the -X blade set.
			stMotionDone[GVL.cXM].trans[stMotionDone[GVL.cXM].ntrans].extTime := stTrack[k].tScanTime;
			stMotionDone[GVL.cXM].trans[stMotionDone[GVL.cXM].ntrans].id := stTrack[k].nHallID;
			stMotionDone[GVL.cXM].trans[stMotionDone[GVL.cXM].ntrans].on := stTrack[k].bEdgeToCompare;
			stMotionDone[GVL.cXM].trans[stMotionDone[GVL.cXM].ntrans].pos := stAxis[GVL.cXM].fHallPosAct;
			stMotionDone[GVL.cXM].ntrans := stMotionDone[GVL.cXM].ntrans +1;
			
			stMotionDone[GVL.cXM].samples[stMotionDone[GVL.cXM].nsamples].extTime := taskStartExtTime[iTimeBuffer];
			stMotionDone[GVL.cXM].samples[stMotionDone[GVL.cXM].nsamples].pos := stAxis[GVL.cXM].axisRef.NcToPlc.ActPos;
			stMotionDone[GVL.cXM].nsamples := stMotionDone[GVL.cXM].nsamples + 1;
		END_IF
		
	END_IF
END_IF

// +X blade set
IF stAxis[GVL.cXP].axisRef.Status.Moving THEN
	//Compare current sequence with recorded sequence. Update position if match. Positive direction.
	IF stAxis[GVL.cXP].axisRef.status.PositiveDirection AND stAxis[GVL.cXP].stHall[GVL.cDirPos, stAxis[GVL.cXP].nTripCount].nSeq = stTrack[k].nSeqToCompare AND 
			stAxis[GVL.cXP].stHall[GVL.cDirPos, stAxis[GVL.cXP].nTripCount].bEdge = stTrack[k].bEdgeToCompare AND (NOT bGoNextSeq) THEN
		stAxis[GVL.cXP].fHallPosAct := stAxis[GVL.cXP].fHallPosCal[GVL.cDirPos, stAxis[GVL.cXP].nTripCount];
		stAxis[GVL.cXP].nTripCount := stAxis[GVL.cXP].nTripCount + 1;
		//track difference between hall sensor and encoder data at trip point
		stAxis[GVL.cXP].fPosDiffAtTrip := stAxis[GVL.cXP].axisRef.NcToPlc.ActPos - stAxis[GVL.cXP].fHallPosAct;
		stAxis[GVL.cXP].bTrackedFlag:=TRUE;
		bGoNextSeq:=TRUE;
		
		IF bInMotion AND MAIN.outShutterStatus.smState<>E_StatesMaint.Calibrating THEN
			nAxisID:= GVL.cXP;
			// The Hall event belongs to the +X blade set.
			stMotionDone[GVL.cXP].trans[stMotionDone[GVL.cXP].ntrans].extTime := stTrack[k].tScanTime;
			stMotionDone[GVL.cXP].trans[stMotionDone[GVL.cXP].ntrans].id := stTrack[k].nHallID;
			stMotionDone[GVL.cXP].trans[stMotionDone[GVL.cXP].ntrans].on := stTrack[k].bEdgeToCompare;
			stMotionDone[GVL.cXP].trans[stMotionDone[GVL.cXP].ntrans].pos := stAxis[GVL.cXP].fHallPosAct;
			stMotionDone[GVL.cXP].ntrans := stMotionDone[GVL.cXP].ntrans +1;
			
			// We're taking the encoder value from process data for this cycle, so the closest
			// approximation we have to the actual sample time is the time at the start of the cycle.
			stMotionDone[GVL.cXP].samples[stMotionDone[GVL.cXP].nsamples].extTime := taskStartExtTime[iTimeBuffer];
			stMotionDone[GVL.cXP].samples[stMotionDone[GVL.cXP].nsamples].pos := stAxis[GVL.cXP].axisRef.NcToPlc.ActPos;
			stMotionDone[GVL.cXP].nsamples := stMotionDone[GVL.cXP].nsamples + 1;
		END_IF
		
	END_IF
END_IF
END_ACTION

ACTION ACT_TrackingSingle:
// Take encoder samples and compare against Hall transitions when only one blade set is moving.

// +X blade set
IF stAxis[GVL.cXP].axisRef.Status.Moving THEN
	//Compare current sequence with recorded sequence. Update position if match. Positive direction.
	IF stAxis[GVL.cXP].axisRef.status.PositiveDirection AND stAxis[GVL.cXP].stHall[GVL.cDirPos, stAxis[GVL.cXP].nTripCount].nSeq = stTrack[k].nSeqToCompare AND 
			stAxis[GVL.cXP].stHall[GVL.cDirPos, stAxis[GVL.cXP].nTripCount].bEdge = stTrack[k].bEdgeToCompare AND (NOT bGoNextSeq) THEN
		stAxis[GVL.cXP].fHallPosAct := stAxis[GVL.cXP].fHallPosCal[GVL.cDirPos, stAxis[GVL.cXP].nTripCount];
		stAxis[GVL.cXP].nTripCount := stAxis[GVL.cXP].nTripCount + 1;
		//track difference between hall sensor and encoder data at trip point
		stAxis[GVL.cXP].fPosDiffAtTrip := stAxis[GVL.cXP].axisRef.NcToPlc.ActPos - stAxis[GVL.cXP].fHallPosAct;
		stAxis[GVL.cXP].bTrackedFlag:=TRUE;
		bGoNextSeq:=TRUE;
		
		IF bInMotion AND MAIN.outShutterStatus.smState<>E_StatesMaint.Calibrating THEN
			nAxisID:= GVL.cXP;
			// The Hall event belongs to the +X blade set.
			stMotionDone[GVL.cXP].trans[stMotionDone[GVL.cXP].ntrans].extTime := stTrack[k].tScanTime;
			stMotionDone[GVL.cXP].trans[stMotionDone[GVL.cXP].ntrans].id := stTrack[k].nHallID;
			stMotionDone[GVL.cXP].trans[stMotionDone[GVL.cXP].ntrans].on := stTrack[k].bEdgeToCompare;
			stMotionDone[GVL.cXP].trans[stMotionDone[GVL.cXP].ntrans].pos := stAxis[GVL.cXP].fHallPosAct;
			stMotionDone[GVL.cXP].ntrans := stMotionDone[GVL.cXP].ntrans +1;			
			// We're taking the encoder value from process data for this cycle, so the closest
			// approximation we have to the actual sample time is the time at the start of the cycle.
			stMotionDone[GVL.cXP].samples[stMotionDone[GVL.cXP].nsamples].extTime := taskStartExtTime[iTimeBuffer];
			stMotionDone[GVL.cXP].samples[stMotionDone[GVL.cXP].nsamples].pos := stAxis[GVL.cXP].axisRef.NcToPlc.ActPos;
			stMotionDone[GVL.cXP].nsamples := stMotionDone[GVL.cXP].nsamples + 1;
		END_IF
		
	END_IF
	//Compare current sequence with recorded sequence. Update position if match. Negative direction.
	IF stAxis[GVL.cXP].axisRef.status.NegativeDirection AND stAxis[GVL.cXP].stHall[GVL.cDirNeg, stAxis[GVL.cXP].nTripCount].nSeq = stTrack[k].nSeqToCompare AND
			stAxis[GVL.cXP].stHall[GVL.cDirNeg, stAxis[GVL.cXP].nTripCount].bEdge = stTrack[k].bEdgeToCompare AND (NOT bGoNextSeq) THEN
		stAxis[GVL.cXP].fHallPosAct := stAxis[GVL.cXP].fHallPosCal[GVL.cDirNeg, stAxis[GVL.cXP].nTripCount];
		stAxis[GVL.cXP].nTripCount := stAxis[GVL.cXP].nTripCount - 1;		
		//track difference between hall sensor and encoder data at trip point
		stAxis[GVL.cXP].fPosDiffAtTrip := stAxis[GVL.cXP].axisRef.NcToPlc.ActPos - stAxis[GVL.cXP].fHallPosAct;
		stAxis[GVL.cXP].bTrackedFlag:=TRUE;
		bGoNextSeq:=TRUE;
		
		IF bInMotion AND MAIN.outShutterStatus.smState<>E_StatesMaint.Calibrating THEN
			nAxisID:= GVL.cXP;
			// The Hall event belongs to the +X blade set.
			stMotionDone[GVL.cXP].trans[stMotionDone[GVL.cXP].ntrans].extTime := stTrack[k].tScanTime;
			stMotionDone[GVL.cXP].trans[stMotionDone[GVL.cXP].ntrans].id := stTrack[k].nHallID;
			stMotionDone[GVL.cXP].trans[stMotionDone[GVL.cXP].ntrans].on := stTrack[k].bEdgeToCompare;
			stMotionDone[GVL.cXP].trans[stMotionDone[GVL.cXP].ntrans].pos := stAxis[GVL.cXP].fHallPosAct;
			stMotionDone[GVL.cXP].ntrans := stMotionDone[GVL.cXP].ntrans +1;
			
			stMotionDone[GVL.cXP].samples[stMotionDone[GVL.cXP].nsamples].extTime := taskStartExtTime[iTimeBuffer];
			stMotionDone[GVL.cXP].samples[stMotionDone[GVL.cXP].nsamples].pos := stAxis[GVL.cXP].axisRef.NcToPlc.ActPos;
			stMotionDone[GVL.cXP].nsamples := stMotionDone[GVL.cXP].nsamples + 1;
		END_IF
		
	END_IF
END_IF

// -X blade set
IF stAxis[GVL.cXM].axisRef.Status.Moving THEN
	//Compare current sequence with recorded sequence. Update position if match. Positive direction.
	IF stAxis[GVL.cXM].axisRef.status.PositiveDirection AND stAxis[GVL.cXM].stHall[GVL.cDirPos, stAxis[GVL.cXM].nTripCount].nSeq = stTrack[k].nSeqToCompare AND
			stAxis[GVL.cXM].stHall[GVL.cDirPos, stAxis[GVL.cXM].nTripCount].bEdge = stTrack[k].bEdgeToCompare AND (NOT bGoNextSeq) THEN
		stAxis[GVL.cXM].fHallPosAct := stAxis[GVL.cXM].fHallPosCal[GVL.cDirPos, stAxis[GVL.cXM].nTripCount];
		stAxis[GVL.cXM].nTripCount := stAxis[GVL.cXM].nTripCount - 1;	
		//track difference between hall sensor and encoder data at trip point
		stAxis[GVL.cXM].fPosDiffAtTrip := stAxis[GVL.cXM].axisRef.NcToPlc.ActPos - stAxis[GVL.cXM].fHallPosAct;
		stAxis[GVL.cXM].bTrackedFlag:=TRUE;
		bGoNextSeq:=TRUE;
		
		IF bInMotion AND MAIN.outShutterStatus.smState<>E_StatesMaint.Calibrating THEN
			nAxisID:= GVL.cXM;
			// The Hall event belongs to the -X blade set.
			stMotionDone[GVL.cXM].trans[stMotionDone[GVL.cXM].ntrans].extTime := stTrack[k].tScanTime;
			stMotionDone[GVL.cXM].trans[stMotionDone[GVL.cXM].ntrans].id := stTrack[k].nHallID;
			stMotionDone[GVL.cXM].trans[stMotionDone[GVL.cXM].ntrans].on := stTrack[k].bEdgeToCompare;
			stMotionDone[GVL.cXM].trans[stMotionDone[GVL.cXM].ntrans].pos := stAxis[GVL.cXM].fHallPosAct;
			stMotionDone[GVL.cXM].ntrans := stMotionDone[GVL.cXM].ntrans +1;
			
			stMotionDone[GVL.cXM].samples[stMotionDone[GVL.cXM].nsamples].extTime := taskStartExtTime[iTimeBuffer];
			stMotionDone[GVL.cXM].samples[stMotionDone[GVL.cXM].nsamples].pos := stAxis[GVL.cXM].axisRef.NcToPlc.ActPos;
			stMotionDone[GVL.cXM].nsamples := stMotionDone[GVL.cXM].nsamples + 1;
		END_IF
		
	END_IF
	//Compare current sequence with recorded sequence. Update position if match. Negative direction.
	IF stAxis[GVL.cXM].axisRef.status.NegativeDirection AND stAxis[GVL.cXM].stHall[GVL.cDirNeg, stAxis[GVL.cXM].nTripCount].nSeq = stTrack[k].nSeqToCompare AND
			stAxis[GVL.cXM].stHall[GVL.cDirNeg, stAxis[GVL.cXM].nTripCount].bEdge = stTrack[k].bEdgeToCompare AND (NOT bGoNextSeq) THEN
		stAxis[GVL.cXM].fHallPosAct := stAxis[GVL.cXM].fHallPosCal[GVL.cDirNeg, stAxis[GVL.cXM].nTripCount];
		stAxis[GVL.cXM].nTripCount := stAxis[GVL.cXM].nTripCount + 1;	
		//track difference between hall sensor and encoder data at trip point
		stAxis[GVL.cXM].fPosDiffAtTrip := stAxis[GVL.cXM].axisRef.NcToPlc.ActPos - stAxis[GVL.cXM].fHallPosAct;
		stAxis[GVL.cXM].bTrackedFlag:=TRUE;
		bGoNextSeq:=TRUE;
		
		IF bInMotion AND MAIN.outShutterStatus.smState<>E_StatesMaint.Calibrating THEN
			nAxisID:= GVL.cXM;
			// The Hall event belongs to the -X blade set.
			stMotionDone[GVL.cXM].trans[stMotionDone[GVL.cXM].ntrans].extTime := stTrack[k].tScanTime;
			stMotionDone[GVL.cXM].trans[stMotionDone[GVL.cXM].ntrans].id := stTrack[k].nHallID;
			stMotionDone[GVL.cXM].trans[stMotionDone[GVL.cXM].ntrans].on := stTrack[k].bEdgeToCompare;
			stMotionDone[GVL.cXM].trans[stMotionDone[GVL.cXM].ntrans].pos := stAxis[GVL.cXM].fHallPosAct;
			stMotionDone[GVL.cXM].ntrans := stMotionDone[GVL.cXM].ntrans +1;
			
			stMotionDone[GVL.cXM].samples[stMotionDone[GVL.cXM].nsamples].extTime := taskStartExtTime[iTimeBuffer];
			stMotionDone[GVL.cXM].samples[stMotionDone[GVL.cXM].nsamples].pos := stAxis[GVL.cXM].axisRef.NcToPlc.ActPos;
			stMotionDone[GVL.cXM].nsamples := stMotionDone[GVL.cXM].nsamples + 1;
		END_IF
		
	END_IF
END_IF
END_ACTION

END_FUNCTION_BLOCK

// ---- POUs/F_MioExtTime.TcPOU
FUNCTION F_MioExtTime : T_DCTIME64
VAR_INPUT
	hallId: DINT;  // The ID number of the Hall sensor that caused the event.
	eventTime: ULINT;  // The timestamp recorded by the MIO.
	iCurTime: INT;  // The index of the current cycle's times in the time buffer.
	taskStartExtTime: T_TaskStartTimes;  // Time buffer. Saved task start times.
	mioSysTime: T_MioSysTimes;  // Time buffer. Saved MIO SysTime values.
END_VAR
VAR CONSTANT
	rolloverCorrection: ULINT := 16#00000001_00000000;
END_VAR
VAR
	iPrevTime: INT;  // The index of the oldest times in the time buffer.
	mioId: DINT;  // 0=MIO-00, 1=MIO-01.
	prevSysTime: ULINT;  // The oldest value of SysTime for the right MIO.
	elapsedTime: ULINT;  // Time between the event and prevSysTime.
END_VAR

// Converts a 32-bit MIO timestamp into a 64-bit external timestamp in T_DCTIME64 format.

// Assume that the MIO timestamp was created sometime between the start of the oldest cycle in the time buffer
// and the current cycle.

// Find out how much time passed on the MIO clock between the oldest cycle
// and the Hall event. Take into account a possible rollover
// of the MIO SysTime.
mioId := hallId / GVL.cFirstMio1Hall;

iPrevTime := (iCurTime + 1) MOD GVL.cTimeBufferDepth;
prevSysTime := mioSysTime[iPrevTime][mioId];
IF eventTime <= prevSysTime THEN
	elapsedTime := (eventTime + rolloverCorrection) - prevSysTime;
ELSE
	elapsedTime := eventTime - prevSysTime;
END_IF

// Assume that the MIO clock and the PLC task clock are running at the same rate.
// Then the external time for the event is just the elapsed time on the MIO
// clock added to the external time at the start of the oldest cycle in the time buffer.
F_MioExtTime := taskStartExtTime[iPrevTime] + elapsedTime;

END_FUNCTION

// ---- POUs/F_HaveDifferentIDs.TcPOU
FUNCTION F_HaveDifferentIDs : BOOL
VAR_INPUT
    msg1: ST_MsgToPLC;
    msg2: ST_MsgToPLC;
END_VAR

(* First compare the fields most likely to have changed. *)
F_HaveDifferentIDs :=
    (msg1.dtime 	<> msg2.dtime) OR_ELSE
    (msg1.sequence 	<> msg2.sequence) OR_ELSE
    (msg1.lowUUID 	<> msg2.lowUUID) OR_ELSE
    (msg1.highUUID	<> msg2.highUUID);

END_FUNCTION

// ---- POUs/StateMachine/FB_Cycler.TcPOU
FUNCTION_BLOCK FB_Cycler
VAR_IN_OUT
	stAxis  : ARRAY [GVL.cXP .. GVL.cXM] OF ST_AxisGroup;
	bTopEntry	: BOOL;	
END_VAR
VAR_INPUT
	stopRequest : BOOL;
	bMotionDone : BOOL;
END_VAR
VAR
	//state-machine
	nCurrentState	: INT;
	nNextState		: INT;
	bLowerEntry		: BOOL;
	tExpoTime		: TIME := T#1S; //change this to desired time
	fSpeed			: LREAL := 0; //change this to desired speed

END_VAR

///////////////////////////////////////////////////////
//Performs open/close motion until commanded to stop.//
//Only USED ON PROTOTYPE							 //
///////////////////////////////////////////////////////
IF bTopEntry = TRUE THEN
	bTopEntry := FALSE;
	nNextState := 3010;
END_IF	
IF nCurrentState <> nNextState THEN
	bLowerEntry := TRUE;
END_IF
nCurrentState := nNextState

CASE nCurrentState OF

	3010: 
		GVL.fbWaitTimer(IN:=TRUE, PT:=tExpoTime);
		stAxis[GVL.cXM].mcMoveAbs(Axis:=stAxis[GVL.cXM].axisRef, Position:= GVL.cPosEnd, Velocity:=fSpeed, Execute:=TRUE);
		IF GVL.fbWaitTimer.Q THEN
			stAxis[GVL.cXP].mcMoveAbs(Axis:=stAxis[GVL.cXP].axisRef, Position:= GVL.cPosEnd, Velocity:=fSpeed, Execute:=TRUE);
		END_IF
		IF stAxis[GVL.cXP].mcMoveAbs.Done AND stAxis[GVL.cXM].mcMoveAbs.Done THEN
			GVL.strokeXP := GVL.strokeXP + 1;
			GVL.strokeXM := GVL.strokeXM + 1;
			GVL.fbWaitTimer(IN:=FALSE);
			stAxis[GVL.cXP].mcMoveAbs(Axis:=stAxis[GVL.cXP].axisRef, Execute:=FALSE);
			stAxis[GVL.cXM].mcMoveAbs(Axis:=stAxis[GVL.cXM].axisRef, Execute:=FALSE);
			nNextState:=3020;
		END_IF
		
	3020:
		GVL.fbWaitTimer(IN:=TRUE, PT:=T#100MS,);
		IF GVL.fbWaitTimer.Q THEN
			GVL.fbWaitTimer(IN:=FALSE);
			IF stopRequest THEN
				stopRequest:=FALSE;
				nNextState:=3999;
			ELSE
				nNextState:=3030;
			END_IF
		END_IF
		
	3030: 
		GVL.fbWaitTimer(IN:=TRUE, PT:=tExpoTime);
		stAxis[GVL.cXP].mcMoveAbs(Axis:=stAxis[GVL.cXP].axisRef, Position:= GVL.cPosStart, Velocity:=fSpeed, Execute:=TRUE);
		IF GVL.fbWaitTimer.Q THEN
			stAxis[GVL.cXM].mcMoveAbs(Axis:=stAxis[GVL.cXM].axisRef, Position:= GVL.cPosStart, Velocity:=fSpeed, Execute:=TRUE);
		END_IF
		IF stAxis[GVL.cXP].mcMoveAbs.Done AND stAxis[GVL.cXM].mcMoveAbs.Done THEN
			GVL.strokeXP := GVL.strokeXP + 1;
			GVL.strokeXM := GVL.strokeXM + 1;
			GVL.fbWaitTimer(IN:=FALSE);
			stAxis[GVL.cXP].mcMoveAbs(Axis:=stAxis[GVL.cXP].axisRef, Execute:=FALSE);
			stAxis[GVL.cXM].mcMoveAbs(Axis:=stAxis[GVL.cXM].axisRef, Execute:=FALSE);
			nNextState:=3040;
		END_IF	
		
	3040:
		GVL.fbWaitTimer(IN:=TRUE, PT:=T#100MS,);
		IF GVL.fbWaitTimer.Q THEN
			GVL.fbWaitTimer(IN:=FALSE);
			IF stopRequest THEN
				stopRequest:=FALSE;
				nNextState:=3999;
			ELSE
				nNextState:=3010;
			END_IF
		END_IF

		
	3999: //End action
		nNextState := 0;
		bMotionDone := TRUE;
END_CASE

END_FUNCTION_BLOCK

// ---- GlobalTextList.TcGTLO
TEXTLIST GlobalTextList
  879 = '                Low Limits                                                High Limits'
  769 = '             Low Limits                                                High Limits'
  522 = '           Low Limits                                                High Limits'
  74 = '           Low Limits                                               High Limits'
  9 = '%7.1f'
  12 = '%7.4f'
  13 = '%7.4f mm'
  8 = '%8.1f'
  53 = '%b'
  52 = '%d'
  4 = '%s'
  16 = '10'
  30 = '1666.6'
  1 = 'Abort'
  25 = 'AxisXP move to:'
  960 = 'AXIS_0: %7.4f mm'
  14 = 'AXIS_1: %7.4f mm'
  15 = 'AXIS_2: %7.4f mm'
  58 = 'Brakes DISENAGAGE'
  10 = 'Brakes ENGAGE'
  11 = 'Brakes RELEASE'
  39 = 'Calibrate'
  28 = 'Close towards X+'
  29 = 'Close towards X-'
  62 = 'CloseShutter'
  33 = 'Continue'
  17 = 'Cycler Task'
  57 = 'EnableAxis'
  68 = 'EnableOutCtrl'
  59 = 'Execute Motion'
  60 = 'GoToProd'
  19 = 'Home'
  22 = 'Home AxisXM'
  21 = 'Home AxisXP'
  23 = 'Home Both'
  34 = 'Home Routine'
  20 = 'home2'
  47 = 'Init'
  311 = 'Low Limits                                                High Limits'
  588 = 'Low Limits                                            High Limits'
  36 = 'Motion Control'
  55 = 'MoveAxisAbsolute'
  32 = 'Normal Visit'
  27 = 'Open Position'
  61 = 'OpenShutter'
  56 = 'Permit'
  65 = 'ProdSpeed'
  0 = 'Reset'
  35 = 'sad'
  5 = 'Set acceleration'
  51 = 'Set Axis'
  54 = 'Set dtime'
  66 = 'Set Exposure'
  7 = 'Set exposure time'
  50 = 'Set Position'
  64 = 'Set ProdSpeed'
  6 = 'Set speed'
  26 = 'Set Speed'
  40 = 'Set Time'
  31 = 'Set Velocity'
  38 = 'Set Velocity%7.1f'
  37 = 'Set Velocity: %7.1f'
  2 = 'Start'
  42 = 'START CYCLER'
  49 = 'State:'
  24 = 'State: %s'
  43 = 'StateLVL1: %s'
  44 = 'nLocalState: %s'
  48 = 'StateLVL2: %s'
  3 = 'Stop'
  41 = 'STOP CYCLER'
  46 = 'Take Exposure'
  63 = 'TakeExposure'
  18 = 'TestMotion Task'
  67 = 'ToggleTestOut'
  45 = 'Travelling Slit'
END_TEXTLIST

// ---- VISUs/Visualization.TcVIS
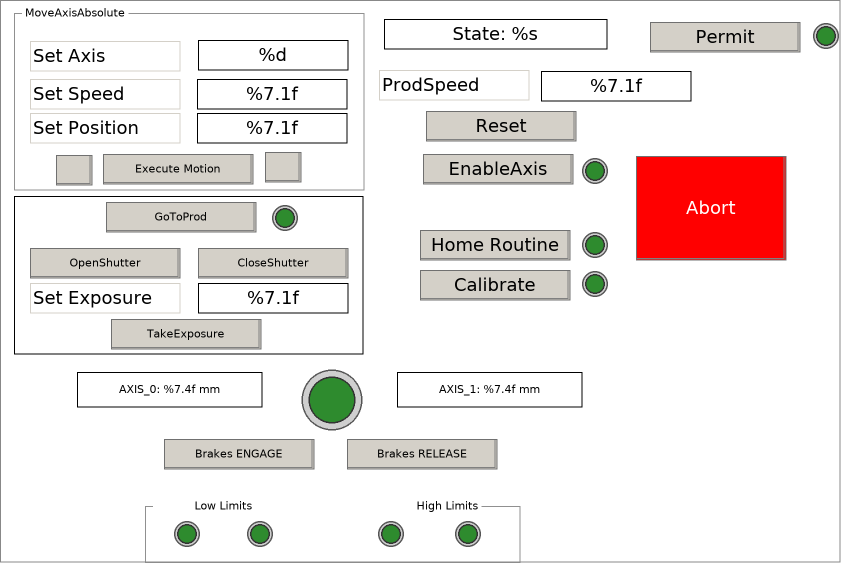
VISUALIZATION Visualization  // 841x563
    Rectangle (14,196 349x158)
    GroupBox (14,5 350x185), "MoveAxisAbsolute"
        Textfield (16,74 150x30), "Set Speed"
            OnMouseUp: write MAIN.inMoveAxisAbsolute.speed via Default, min 0, max 1667, format %7.1f
        Rectangle (183,74 150x30), "%7.1f", text variable: MAIN.inMoveAxisAbsolute.speed
        Textfield (16,108 150x30), "Set Position"
            OnMouseUp: write MAIN.inMoveAxisAbsolute.position via Default, min 0, max 751, format %7.1f
        Rectangle (183,108 150x30), "%7.1f", text variable: MAIN.inMoveAxisAbsolute.position
        Button (89,149 150x30), "Execute Motion"
            OnMouseUp: execute { MAIN.inMoveAxisAbsolute.dtime := MAIN.inMoveAxisAbsolute.dtime + 1; }
        Button (251,147 36x30)
            OnMouseUp: execute { MAIN.inMoveAxisAbsolute.position:=750.76; }
        Button (42,150 36x30)
            OnMouseUp: execute { MAIN.inMoveAxisAbsolute.position:=0; }
    Button (347,439 150x30), "Brakes RELEASE"
        OnMouseDown: execute {
            MAIN.inChangeBrakeState.axisIndex := 0;
            MAIN.inChangeBrakeState.state := FALSE;
            MAIN.inChangeBrakeState.dtime := MAIN.inChangeBrakeState.dtime + 1;
        }
        OnMouseUp: execute {
            MAIN.inChangeBrakeState.axisIndex := 1;
            MAIN.inChangeBrakeState.state := FALSE;
            MAIN.inChangeBrakeState.dtime := MAIN.inChangeBrakeState.dtime + 1;
        }
    Lamp1 (297,365 70x70), variable: (MAIN.stAxis[0].bBrake and MAIN.stAxis[1].bBrake), style: Lamp-Lamp1-Green
    Rectangle (77,372 185x35), "AXIS_0: %7.4f mm", text variable: MAIN.stAxis[0].axisRef.NcToPlc.ActPos
    Rectangle (397,372 185x35), "AXIS_1: %7.4f mm", text variable: MAIN.stAxis[1].axisRef.NcToPlc.ActPos
    Button (426,111 150x30), "Reset"
        OnMouseUp: execute { MAIN.inReset.dtime := MAIN.inReset.dtime + 1; }
    Button (636,156 150x104), "Abort"
        OnMouseUp: execute { MAIN.inReset.dtime := MAIN.inReset.dtime + 1; }
    Rectangle (384,19 223x30), "State: %s", text variable: MAIN.outShutterStatus.smState
    Button (420,230 150x30), "Home Routine"
        OnMouseUp: execute { MAIN.inHomeAxis.dtime := MAIN.inHomeAxis.dtime + 1; }
    Textfield (30,41 150x30), "Set Axis"
        OnMouseUp: write MAIN.inMoveAxisAbsolute.axisIndex via Default, min 0, max 1, format %b
    Rectangle (198,40 150x30), "%d", text variable: MAIN.inMoveAxisAbsolute.axisIndex
    Lamp1 (580,230 30x30), variable: MAIN.stAxis[0].axisRef.Status.Homed and MAIN.stAxis[1].axisRef.Status.Homed, style: Lamp-Lamp1-Green
    Button (420,270 150x30), "Calibrate"
        OnMouseUp: execute { MAIN.inCalibrate.dtime := MAIN.inCalibrate.dtime + 1; }
    Button (164,439 150x30), "Brakes ENGAGE"
        OnMouseDown: execute {
            MAIN.inChangeBrakeState.axisIndex := 0;
            MAIN.inChangeBrakeState.state := TRUE;
            MAIN.inChangeBrakeState.dtime := MAIN.inChangeBrakeState.dtime + 1;
        }
        OnMouseUp: execute {
            MAIN.inChangeBrakeState.axisIndex := 1;
            MAIN.inChangeBrakeState.state := TRUE;
            MAIN.inChangeBrakeState.dtime := MAIN.inChangeBrakeState.dtime + 1;
        }
    Button (650,22 150x30), "Permit"
        OnMouseDown: execute { MAIN.bAuxElxPermit := NOT MAIN.bAuxElxPermit; }
    Lamp1 (811,21 30x30), variable: MAIN.bAuxElxPermit, style: Lamp-Lamp1-Green
    Button (423,154 150x30), "EnableAxis"
        OnMouseUp: execute { MAIN.inEnableAllAxes.dtime := MAIN.inEnableAllAxes.dtime + 1; }
    Button (106,202 150x30), "GoToProd"
        OnMouseUp: execute { MAIN.inGoToProd.dtime := MAIN.inGoToProd.dtime + 1; }
    Button (30,248 150x30), "OpenShutter"
        OnMouseUp: execute { MAIN.inOpenShutter.dtime := MAIN.inOpenShutter.dtime + 1; }
    Button (198,248 150x30), "CloseShutter"
        OnMouseUp: execute { MAIN.inCloseShutter.dtime := MAIN.inCloseShutter.dtime + 1; }
    Button (111,319 150x30), "TakeExposure"
        OnMouseUp: execute { MAIN.inTakeExposure.dtime := MAIN.inTakeExposure.dtime + 1; }
    Rectangle (541,71 150x30), "%7.1f", text variable: MAIN.inReset.speed
    Textfield (379,70 150x30), "ProdSpeed"
        OnMouseUp: write MAIN.inReset.speed via Default, min 0, max 1667, format %7.1f
    Textfield (30,283 150x30), "Set Exposure"
        OnMouseUp: write MAIN.inTakeExposure.exposureTime via Default, min 100, format %7.1f
    Rectangle (198,283 150x30), "%7.1f", text variable: MAIN.inTakeExposure.exposureTime
    Lamp1 (580,269 30x30), variable: MAIN.stAxis[0].bIsCalibrated and MAIN.stAxis[1].bIsCalibrated;, style: Lamp-Lamp1-Green
    Lamp1 (580,156 30x30), variable: MAIN.outShutterStatus.axis[0].enabled and MAIN.outShutterStatus.axis[1].enabled;, style: Lamp-Lamp1-Green
    Lamp1 (172,519 30x30), variable: MAIN.stAxis[0].bLimitHome;, style: Lamp-Lamp1-Green
    Lamp1 (245,519 30x30), variable: MAIN.stAxis[1].bLimitDeployed;, style: Lamp-Lamp1-Green
    Lamp1 (376,519 30x30), variable: MAIN.stAxis[0].bLimitDeployed;, style: Lamp-Lamp1-Green
    Lamp1 (453,519 30x30), variable: MAIN.stAxis[1].bLimitHome;, style: Lamp-Lamp1-Green
    GroupBox (145,498 375x65), "Low Limits High Limits"
    Lamp1 (270,203 30x30), variable: MAIN.fbShutterSM.fbEnabled.bShutterReady;, style: Lamp-Lamp1-Green
END_VISUALIZATION
